// TIA Portal V16 export
// export: Created 2022-02-28T20:45:46.9136373Z, ExportSetting WithDefaults, DisplayName Totally Integrated Automation Portal, DisplayVersion V16, DisplayName TIA Portal Version Control Interface, DisplayVersion V16, DisplayName TIA Portal Openness, DisplayVersion V16, DisplayName STEP 7 Professional, DisplayVersion V16, DisplayName STEP 7 Safety, DisplayVersion V16, DisplayName WinCC Advanced, DisplayVersion V16
DATA_BLOCK "DataMan_DB"   // DB9
VERSION : 0.1
// stored: AutoNumber true, DBAccessibleFromOPCUA true, InstanceOfName DataMan, InstanceOfType FB
"DataMan"
   // VAR_OUTPUT
   //    DataMan_Trigger_Ready : Bool;
   //    DataMan_TriggerAck : Bool;
   //    DataMan_ResultAvailable : Bool;
   //    DataMan_ResultID : Word;
   //    "DataMan Result Code" : Word;
   //    "DataMan Result Length" : Word;
   //    ResultData : Array[0..63] of Byte;
   // END_VAR
   // VAR_IN_OUT
   //    DataMan_Trigger_Enable : Bool;
   //    DataMan_Trigger : Bool;
   //    DataMan_ResultsAck : Bool;
   // END_VAR
   // VAR
   //    Resultado_Pendiente : Bool;
   //    "Lastest Result" : Struct
   //       ID : Int;
   //       Flags : Int;
   //       Lenght : Int;
   //       Value : Array[0..63] of Byte;
   //    END_STRUCT;
   // END_VAR
BEGIN
END_DATA_BLOCK
